{attribute 'qualified_only'}
VAR_GLOBAL CONSTANT
		CstNbAOEntries			: INT :=  50 ;
END_VAR

(* stored: Version 1.1.0.1, ProductVersion 3.1.4024.6
   GVL GVL_Cst: Id {fe9331df-1340-4161-a816-d54d4e661e7b} *)
